VAR_GLOBAL
// Включение второй скорости для секций

bDrive4s01Speed2			AT%Q* :BOOL;

bDrive4s02Speed2			AT%Q* :BOOL;

bDrive4s03Speed2			AT%Q* :BOOL;

bDrive4s04Speed2			AT%Q* :BOOL;

bDrive4s05Speed2			AT%Q* :BOOL;

bDrive4s06Speed2			AT%Q* :BOOL;
END_VAR

(* stored: Version 1.1.0.1, ProductVersion 3.1.4024.3
   GVL GVL_bDriveSpeed_4: Id {6a642211-04f6-4ccb-b824-0d27be70e849} *)
